FUNCTION_BLOCK FB_CommandProcess

// Parameters of receiving and transferring data
VAR
	mInputData  	AT%I* : ARRAY[0..MAX_BUFFER_LENGTH-1] OF MotionCommand; //array stores data form host machine 
	mOutputData  	AT%Q* : MotionCommand; //data read from buffer  
	
	iReadIndex AT%Q* : UDINT := 0; // sum of sent data
	iWriteIndex AT%I* : UDINT := 0; // sum of received data
	localReadIndex : UDINT := 0;
END_VAR

;

METHOD mInitialize : BOOL
VAR_INPUT
END_VAR
// Wait for host machine to fill command buffer;
mInitialize := FALSE;
iReadIndex := 0;
localReadIndex := 0;

// The buffer is filled for the first time
IF iWriteIndex = GlobalVar.MAX_BUFFER_LENGTH THEN
	mInitialize := TRUE;
END_IF
END_METHOD

METHOD mReset : BOOL
VAR_INPUT
END_VAR
mReset := TRUE;

iReadIndex := 0;
localReadIndex := 0;
MEMSET(ADR(mOutputData), 0, SIZEOF(MotionCommand));

mReset := FALSE;
END_METHOD

METHOD mSendCommand : BOOL
VAR_INPUT
END_VAR
// Link mOutputdata to corresponding data structure in Cpp module
mSendCommand := FALSE;

IF iReadIndex < iWriteIndex  THEN
	
	mOutputData := mInputData[localReadIndex];

	iReadIndex := iReadIndex + 1;
	
	localReadIndex := (iReadIndex AND GlobalVar.BUFFER_MASK);
			
	mSendCommand := TRUE;
END_IF
END_METHOD

END_FUNCTION_BLOCK

(* stored: Version 1.1.0.1
   POU FB_CommandProcess: Id {4cc609f8-5b4e-4130-af29-e2e869c45ddc}, SpecialFunc None
   Method mInitialize: Id {3cbcc8bb-c0f0-4bab-bdd7-b42a91bdb277}
   Method mReset: Id {79b35ea7-30e4-400c-b6ef-7774d6fe749b}
   Method mSendCommand: Id {0ba57674-b202-417a-8c41-1345aa1012c0} *)
